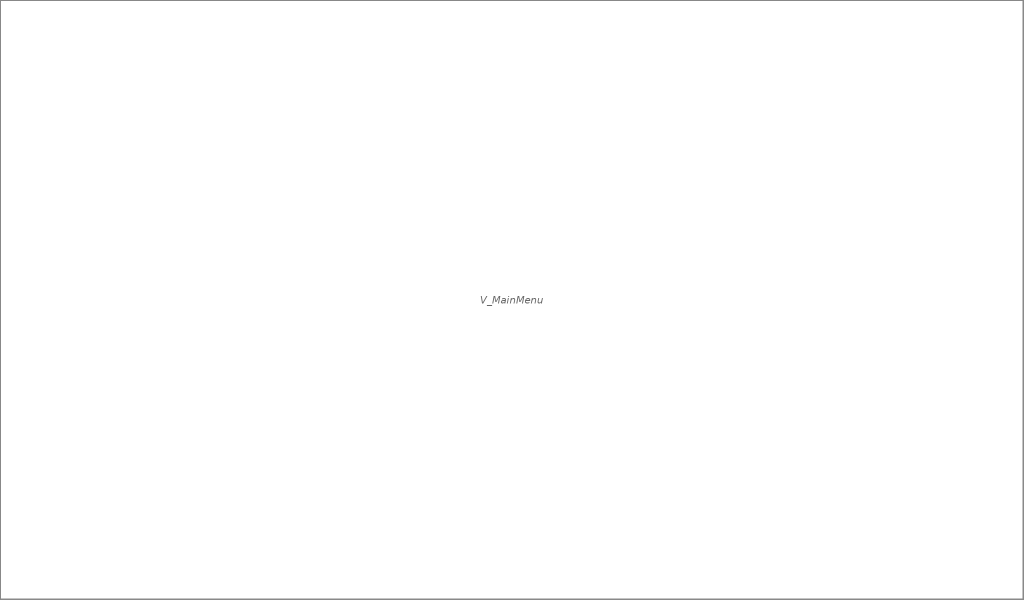
VISUALIZATION V_Main  // 1024x600
    Frame (0,0 1024x600), frame switch variable: GVL_HMI.ShowProductionPopup
        shows V_MainMenu(HMI := MAIN.Seedra.PackMLBaseModule_HMI, HMIAxeX := MAIN.Seedra.GantryXYZ.AxisX.AxisBase_HMI, HMI_Recipe := MAIN.Seedra.RecipeConfig_HMI)
        shows V_InfoMenu()
END_VISUALIZATION

(* stored: Version 1.1.0.1, ProductVersion 3.1.4024.15
   Visu V_Main: Id {60cc94dd-423f-42a7-ac12-2e8b2f9f36e1} *)
